// TIA Portal V19 export
FUNCTION "PTrk_Presence" : Void   // FC112, LAD
// stored: Access Published, SetENOAutomatically false
   VAR_INPUT
      Item : "PTrk_Item";
   END_VAR
BEGIN

REGION Network 1 (SCL)
   ENO := #Item.P_ID <> 0;
END_REGION
END_FUNCTION
